DEVICE_TYPE BeagleBoneBlack (* BeagleBoneBlack controller *)
  (* Standard: 61499 ITA; Description: Remotely Managed Device *)
  (* Version 1.0, 2015-10-31, Alois Zoitl, fortiss GmbH, Initial version *)
  VAR_INPUT
    MGR_ID : WSTRING := "localhost:61499"; (* Device manager socket ID *)
  END_VAR
END_DEVICE_TYPE
